// LS Electric XG5000 project: 동남139
// PLC NewPLC
// module base 0 slot 0: 입출력 모듈:XBC-DN/DP14E (DC 24V 입력 8점, 트랜지스터 출력 6점)

PROGRAM NewProgram (task: 스캔 프로그램)

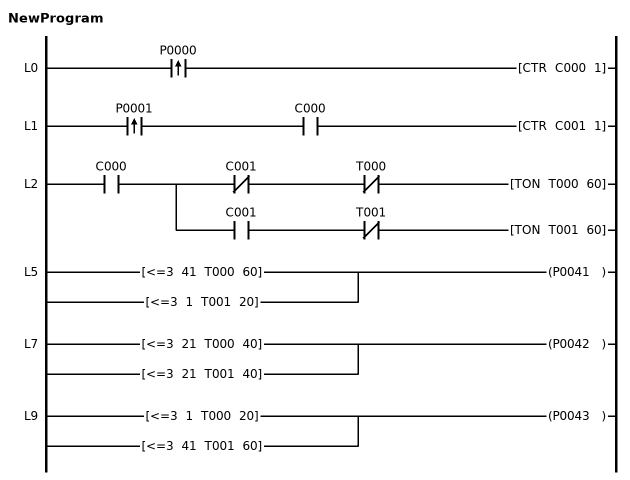
; L0
LOADP     P0000
CTR       C000 1
; L1
LOADP     P0001
AND       C000
CTR       C001 1
; L2
LOAD      C000
MPUSH
AND NOT   C001
AND NOT   T000
TON       T000 60
MPOP
AND       C001
AND NOT   T001
TON       T001 60
; L5
LOAD<=3   41 T000 60
OR<=3     1 T001 20
OUT       P0041
; L7
LOAD<=3   21 T000 40
OR<=3     21 T001 40
OUT       P0042
; L9
LOAD<=3   1 T000 20
OR<=3     41 T001 60
OUT       P0043